FUNCTION_BLOCK StringBuilderExtBuffer
VAR
	_Buffer : __SYSTEM.AnyType;
	_Length : DINT;
END_VAR

METHOD Append : REFERENCE TO StringBuilderExtBuffer
VAR_INPUT
	value : T_MaxString;
END_VAR
VAR
	lengthToCopy : DINT;
END_VAR
lengthToCopy := LIMIT(
	DINT#0, 								// min
	LEN(value), 							// value
	(_Buffer.diSize - TO_DINT(_Length) - 1) // max
);

MEMCPY(
	destAddr := _Buffer.pValue + _Length,
	srcAddr := ADR(value),
	n := lengthToCopy
);

_Length := _Length + lengthToCopy;

Append := THIS^;
END_METHOD

METHOD AppendByPointer : REFERENCE TO StringBuilderExtBuffer
VAR_INPUT
	value : POINTER TO STRING;
END_VAR
VAR
	valueLength : DINT;
	lengthToCopy : DINT;
END_VAR
valueLength := LEN2(value);

lengthToCopy := LIMIT(
	DINT#0, 								// min
	valueLength, 							// value
	(_Buffer.diSize - TO_DINT(_Length) - 1) // max
);

MEMCPY(
	destAddr := _Buffer.pValue + _Length,
	srcAddr := value,
	n := lengthToCopy
);

_Length := _Length + lengthToCopy;

AppendByPointer := THIS^;
END_METHOD

{attribute 'monitoring' := 'call'}
PROPERTY Buffer : REFERENCE TO __SYSTEM.AnyType
GET
Buffer REF= _Buffer;
END_GET
END_PROPERTY

METHOD Clear : REFERENCE TO StringBuilderExtBuffer
MEMSET(
	destAddr := _Buffer.pValue,
	fillByte := 0,
	n := _Buffer.diSize
);

_Length := 0;

Clear := THIS^;
END_METHOD

METHOD FB_init : BOOL
VAR_INPUT
	bInitRetains : BOOL; // if TRUE, the retain variables are initialized (warm start / cold start)
	bInCopyCode : BOOL;  // if TRUE, the instance afterwards gets moved into the copy code (online change)
	
	buffer : ANY;
END_VAR
_Buffer := buffer;

_Length := LEN2(pSTRING := buffer.pValue);
END_METHOD

PROPERTY IsEmpty : BOOL
GET
IsEmpty := Length = 0;
END_GET
END_PROPERTY

{attribute 'monitoring' := 'call'}
PROPERTY Length : DINT
GET
Length := _Length;
END_GET
END_PROPERTY

METHOD SetBuffer : REFERENCE TO StringBuilderExtBuffer
VAR_INPUT
	buffer : ANY;
END_VAR
_Buffer := buffer;

_Length := LEN2(pSTRING := buffer.pValue);
END_METHOD

END_FUNCTION_BLOCK

(* stored: Version 1.1.0.1, ProductVersion 3.1.4024.12
   POU StringBuilderExtBuffer: Id {261b6625-c824-4ba7-8b30-9e72c2ea80b1}, SpecialFunc None
   Method Append: Id {938d36be-8533-462c-9d1d-ce287c37acd6}
   Method AppendByPointer: Id {301900e5-220a-47d4-9de7-16c47b9c4624}
   Property Buffer: Id {49532420-43d6-4129-898d-64af45bb5d78}
   Get Get: Id {c541380c-ae02-499c-aa5c-41269e7cc87d}
   Method Clear: Id {51ab4961-e81a-4543-af50-292474c11adf}
   Method FB_init: Id {1cd4845e-24ab-4b4d-827c-8967da5ce213}
   Property IsEmpty: Id {a1bfbe9c-c914-4227-bc67-942558ab1b1e}
   Get Get: Id {54abde92-1704-48e1-87d6-d4e40dd27319}
   Property Length: Id {96473c69-e45d-4c53-b3ac-0d60f1275aaa}
   Get Get: Id {a114f96d-8619-4574-ab93-f9c3d8b011c8}
   Method SetBuffer: Id {604f339c-820d-4f30-abfa-03379d2adc39} *)
